Staubli VAL3: sendStatus.pgx

public program sendStatus()
  local num l_nRetVal
begin
    call sendData(siTcpIpFbk, rosStatusMsg.prefix.nData, nDataOut)
    call sendData(siTcpIpFbk, rosStatusMsg.header.nData, nDataOut)
    call sendData(siTcpIpFbk, rosStatusMsg.body.nData, nDataOut)
end
